# EPICS substitutions: mv2/mv2App/Db/user.substitutions
# Example substitutions file

file "db/dbExample1.db" {
    { user = "rory" }
}

file db/dbExample2.db {
    pattern { user, no, scan }
        { "rory", 1, "1 second" }
        { "rory", 2, "2 second" }
        { "rory", 3, "5 second" }
}
